FUNCTION_BLOCK "FB_TimerOnOffDelay"
TITLE = FB_TimerOnOffDelay
{ S7_Optimized_Access := 'TRUE' }
AUTHOR : MHSE
FAMILY : GeneralSystemFunctions
VERSION : 3.0
// ATTRIBUTES
// AUTO_NUMBER = True
// BLOCK_NUMBER = 32
// END_ATTRIBUTES
//Function block to generate on/off signal delay.
   VAR_INPUT
      iudi_OnDelayTime { ExternalAccessible := 'False'; ExternalVisible := 'False'; ExternalWritable := 'False'} : UDInt;   // On delay time [ms]
      iudi_OffDelayTime { ExternalAccessible := 'False'; ExternalVisible := 'False'; ExternalWritable := 'False'} : UDInt;   // Off delay time [ms]
      ix_SignalToDelay { ExternalAccessible := 'False'; ExternalVisible := 'False'; ExternalWritable := 'False'} : Bool;   // Input signal to be delayed
      ix_Enable { ExternalAccessible := 'False'; ExternalVisible := 'False'; ExternalWritable := 'False'} : Bool := TRUE;   // Timer Enable
   END_VAR

   VAR_OUTPUT
      qlr_ActualTime { ExternalAccessible := 'False'; ExternalVisible := 'False'; ExternalWritable := 'False'} : LReal;   // Actual time
      qx_DelayedSignal { ExternalAccessible := 'False'; ExternalVisible := 'False'; ExternalWritable := 'False'} : Bool;   // Delayed signal output
   END_VAR

   VAR
      s_R_TRIG_Signal {InstructionName := 'R_TRIG'; LibVersion := '1.0'; ExternalAccessible := 'False'; ExternalVisible := 'False'; ExternalWritable := 'False'; S7_SetPoint := 'False'} : R_TRIG;   // Siemens "R_Trig" - to prepare the rising edge trigger on "ix_SignalToDelay" signal
      s_F_TRIG_Signal {InstructionName := 'F_TRIG'; LibVersion := '1.0'; ExternalAccessible := 'False'; ExternalVisible := 'False'; ExternalWritable := 'False'; S7_SetPoint := 'False'} : F_TRIG;   // Siemens "F_Trig" - to prepare the falling edge trigger on "ix_SignalToDelay" signal
   END_VAR
   VAR RETAIN
      slr_ActualDelayTime { ExternalAccessible := 'False'; ExternalVisible := 'False'; ExternalWritable := 'False'} : LReal;   // Actual delay time [ms]
   END_VAR


BEGIN
	(*
	----------------------------------------------------------------------------------------

	Version history:
	Date        | Version   | Author        | Remark
	----------------------------------------------------------------------------------------
	24/05/2019  | 0.1       | L.Klar        | first release MHS TIA 15.1
	24/07/2019  | 2.0       | L.Klar        | 2.0 MHS library release TIA 15.1
	26/08/2019  | 2.1       | M.Kurpiers    | Comments adjusted
	04/11/2019  | 2.2       | L.Klar        | Prevoius cycle scan changed from memory to DB variable
	12/11/2019  | 3.0       | P.Majka       | 3.0 MHS library release TIA 15.1
	21/02/2023  | 4.0       | F.Baten       | 4.0 Release TIA 17.5
	*)

	REGION Step 1 – Input signal edge detection

	    #s_R_TRIG_Signal(CLK := #ix_SignalToDelay);


	    #s_F_TRIG_Signal(CLK := #ix_SignalToDelay);

	END_REGION

	REGION Step 2 – Actual delay time initialization

	    IF (#s_R_TRIG_Signal.Q OR #s_F_TRIG_Signal.Q)           // Input signal changed
	    THEN

	        #slr_ActualDelayTime := 0;

	    END_IF;

	END_REGION

	REGION Step 3 – On/Off delay time calculation


	    IF (#ix_SignalToDelay                                       // Signal to be delayed is active
	        AND #ix_Enable)                                         // Ttimer enabled
	    THEN

	        // Timer on
	        IF (#slr_ActualDelayTime >= #iudi_OnDelayTime)
	        THEN

	            #qx_DelayedSignal := TRUE;

	        ELSE

	            #slr_ActualDelayTime += "DB_Memory".PrevCycleTime;

	        END_IF;

	    END_IF;

	    // Timer off
	    IF (NOT #ix_SignalToDelay                                   // Signal to delay is not active
	        AND #ix_Enable)                                         // Timer is enabled
	    THEN

	        IF (#slr_ActualDelayTime >= #iudi_OffDelayTime)
	        THEN

	            #qx_DelayedSignal := FALSE;

	        ELSE

	            #slr_ActualDelayTime += "DB_Memory".PrevCycleTime;

	        END_IF;

	    END_IF;

	END_REGION

	REGION Step 4 – Actual time

	    #qlr_ActualTime := #slr_ActualDelayTime;

	END_REGION
END_FUNCTION_BLOCK

